FUNCTION_BLOCK ABSTRACT FB_BaseMotionStage
VAR_INPUT
END_VAR
VAR_OUTPUT
END_VAR
VAR
END_VAR

END_FUNCTION_BLOCK

(* stored: Version 1.1.0.1
   POU FB_BaseMotionStage: Id {47a73cca-a73f-4109-a111-1cbf4727c2fa}, SpecialFunc None *)
